Fanuc KAREL source: kx00005.KL

-- PROVISIONAL review KL for V1013-1; original PC SHA256 8d96dcadced47cded26315a267ec52ee171881f96c7aeecb4b7253048f4c098d
-- Incomplete behavior may be omitted. Consult companion uncertainty JSON. Do not deploy.
PROGRAM KX00005
%NOLOCKGROUP
VAR
  I : INTEGER
  J : INTEGER
  B : BOOLEAN
  F : FILE
  S : STRING[80]
-- UNRESOLVED_DECL P type=000102
BEGIN
  -- UNRESOLVED_PC offsets 5-32; opcodes 22,3F,3F,3D
  -- UNRESOLVED_PC offsets 37-44; opcodes 22,A3
  -- UNRESOLVED_PC offsets 49-56; opcodes 22,39
  -- UNRESOLVED_PC offsets 61-65; opcodes 7F
END KX00005
